PROGRAM prg_GetMinimum
VAR
	FB_GetMinimum: FB_GetMinimum;
	FB_Click_Log: FB_Click_Log;
	bDrukknop		AT		%I*		:BOOL;
	tMinTime		AT		%Q*		:TIME;
	LogTijden 		:ARRAY[1..10] OF TIME;
END_VAR

FB_Click_Log(Drukknop:= bDrukknop, Tijden=> LogTijden);
FB_GetMinimum(Times:= LogTijden, MinTime=> tMinTime);

//Met een functie ipv FunctieBlok (ongetest)
//tMinTime := FGetMinimum(LogTijden);

END_PROGRAM

(* stored: Version 1.1.0.1, ProductVersion 3.1.4024.15
   POU prg_GetMinimum: Id {15009af4-906b-4550-a345-9c273a7df78c}, SpecialFunc None *)
